TYPE ST_SendDpHstData :
STRUCT
	bError		: BOOL;
	bSubsOn		: BOOL;
END_STRUCT
END_TYPE

(* stored: Version 1.1.0.1, ProductVersion 3.1.4024.12
   DUT ST_SendDpHstData: Id {ce41ea38-650d-0515-339c-8cae0e6619cf} *)
